# B&R Automation Studio project AutomatedPongGame (part 5)

#### TonTimer.cpp - Implementation code
```cpp
/********************************************************************
 * COPYRIGHT --
 ********************************************************************
 * Program: TonTimer
 * File: TonTimer.cpp
 ********************************************************************
 * Implementation of program TonTimer
 ********************************************************************/

#include <bur/plctypes.h>
#include <string.h>

#include "..\Timer\Timer.hpp"

/* Heap size for this program */
unsigned long bur_heap_size = 0xFFFF;

#ifdef _DEFAULT_INCLUDES
#include <AsDefault.h>
#endif

#define TRAPPER_BITMASK 0x02
#define KANTELMECHANISME_BITMASK 0x04

DINT getal1;
INT getal2;

void _INIT TonTimerINIT(void)
{
}

void _CYCLIC TonTimerCYCLIC(void)
{
	/* set and reset timer */

	isTrapperButtonPressed = ((digitalInput & TRAPPER_BITMASK) == 0);
	isVeldButtonPressed = ((digitalInput & KANTELMECHANISME_BITMASK) == 0);
	isTrapperButtonNotPressed = !isTrapperButtonPressed;
	isVeldButtonNotPressed = !isVeldButtonPressed;
	/* read output values to process variables */
	/* Cyclic call. This is needed because the TON Function block is used in the class IECTonTimer */
	getal1 = (INT)getal2;
}

void _EXIT TonTimerEXIT(void)
{

}
```

Listed in the project but not available here: Logical/Global.typ, Logical/Libraries/UnitTest/UnitTest/include, Logical/Libraries/Library/Variables.var, Logical/Main/Types.typ, Logical/gAxis01obj/gAxis01a, Logical/gAxis02obj/gAxis02a, Logical/UnitTests/UnitTests/Tests_FieldMotor_C/testSuite.c, Logical/UnitTests/UnitTests/TestSet_Templates/Set_Testcases.c, Logical/UnitTests/UnitTests/TestSet_Templates/Set_SetupTeardown.c, Logical/UnitTests/UnitTests/TestSet_Templates/Set_Complete.c, Logical/UnitTests/UnitTests/Tests_BallControl_C/testSuite.c, Logical/UnitTests/UnitTests/Tests_DistanceSensor_C/testSuite.c, Logical/UnitTests/UnitTests/Tests_FieldControl_C/testSuite.c, Logical/UnitTests/UnitTests/Tests_InclinoSensor_C/testSuite.c, Logical/UnitTests/UnitTests/Tests_PongGame_C/testSuite.c, Logical/UnitTests/HelperTool_Supported/Tests_PaddleMotor_C/testSuite.c, Logical/LibACP10MC_SingleAx_C/Basic/basic.typ, Logical/LibACP10MC_SingleAx_C/Basic/basic.var, Logical/Timer_CPP/Timer/Timer.hpp, Logical/Timer_CPP/Timer/ITimer.hpp, Logical/Timer_CPP/Timer/IECTonTimer.cpp, Logical/Timer_CPP/Timer/IECTofTimer.cpp, Logical/Timer_CPP/Timer/IECTpTimer.hpp, Logical/Timer_CPP/Timer/IECTimerFactory.hpp, Logical/Timer_CPP/Timer/IECTimerFactory.cpp
